FUNCTION_BLOCK R_SYS_T
VAR_INPUT
	It_SynchTime						: TIME; 
END_VAR
VAR_OUTPUT
	Odt_RTCTime						: DT; 
	Odw_Milliseconds					: DWORD; 
	Ox_TimeValid						: BOOL; 
END_VAR
VAR
	So_SynchronizeTimer			: TON; 
	So_ReadSystemTime			: NT_GetTime; 
	Ss_SystemTime					: TIMESTRUCT; 
	Sx_Synch								: BOOL; 
	So_SynchTrigger					: F_TRIG; 
	So_RTC								: RTC_EX; 
	
	//Debug variables
	Si_SynchCounter					: DWORD; 
	
END_VAR

//Defines
{define DEBUG}

//Read System Time cyclic with period based on the Synch time 
So_SynchronizeTimer(IN := NOT So_SynchronizeTimer.Q, PT := It_SynchTime);
So_ReadSystemTime(START := So_SynchronizeTimer.Q,  TMOUT := DEFAULT_ADS_TIMEOUT, TIMESTR => Ss_SystemTime); 

//Create the synchronise bit
So_SynchTrigger(CLK := (So_ReadSystemTime.BUSY AND NOT So_ReadSystemTime.ERR)); 

//Count the Synchs in Debug Mode
{IF defined (DEBUG)}
	IF(So_SynchTrigger.Q) THEN 
		Si_SynchCounter := Si_SynchCounter + 1; 
	END_IF
{END_IF}

//RTC Synchronisieren und auslesen 
So_RTC(EN := So_SynchTrigger.Q, PDT := SYSTEMTIME_TO_DT(Ss_SystemTime), PMSEK := Ss_SystemTime.wMilliseconds, Q => Ox_TimeValid, CDT => Odt_RTCTime, CMSEK => Odw_Milliseconds);

END_FUNCTION_BLOCK

(* stored: Version 1.1.0.1, ProductVersion 3.1.4024.9
   POU R_SYS_T: Id {dd1e5667-3a03-4853-8f36-d7efde7cc85d}, SpecialFunc None *)
